# B&R Automation Studio project mappFramework
Automation Studio 4.12.4.107 SP; technology packages: mapp 5.18.0, mappCockpit 5.18.0, mappMotion 5.18.1, mappView 5.18.1

## Configuration Simulation

CPU PC_any, AutomationRuntime E4.91, Build 6.3.0, Safety 0.0, Vc V4.72.3

### Task classes (Cpu.sw)
```
Cyclic#1 (cycle 10000 us):
  AlarmMgr <- Infrastructure.VC4.AlarmX.AlarmMgr.prg
  AppAxis_1 <- MachineControl.AppAxis_1.AppAxis_1.prg
  AxisMgr <- MachineControl.AxisTemplate.AxisMgr.prg [disabled]
Cyclic#8 (cycle 10000 us):
  BackupMgr <- Infrastructure.VC4.Backup.BackupMgr.prg
  FileMgr <- Infrastructure.VC4.File.FileMgr.prg
  UsbMgr <- Infrastructure.VC4.Usb.UsbMgr.prg  // USB manager
  RecipeMgr <- Infrastructure.VC4.Recipe.RecipeMgr.prg
  UserXMgr <- Infrastructure.VC4.UserX.UserXMgr.prg
  AuditMgr <- Infrastructure.VC4.Audit.AuditMgr.prg
  ReportMgr <- Infrastructure.VC4.Report.ReportMgr.prg
NcDataObjects: McDriveLog
VcDataObjects: mappFr <- VC4.mappFrameworkVisu.dob
Binaries: arsvcreg, mCoWebSc, McProfGen, mcacpdrv, TCLang, arflatprv, FWRules, arcoal, udbdef, mvLoader, TCData, vcfntttf, vcxml, vccbmp, vcshared, vccscale, vcmgr, vccshape, vcfile, vcgclass, vccpiech, arial, vcchspot, vccslider, vcdsint, vccbtn, vccline, vcpfar00, vccovl, vcctext, vcalarm, vcbclass, vcrt, vccnum, vccstr, Visu03, vccddbox, arialbd, vcctrend, vcpdsw, vccpopup, vccurl, vcnet, vcpdvnc, vcdsloc, vcclbox, Visu02, Visu01, vctcal, vcchtml, vccdt, vcpkat, UserXCfg, UserXlogin, arconfig, FileCfg, RecipeXML, TC, RecipeFile, User, AlarmXCfg, asfw, iomap, Role, Axis1Alm, VAppAxis1, ashwd, RecipeCSV, Settings, AppAxis1, BackupCfg, ashwac, AlarmXHist, sysconf, Axis1Grp, BackupFile, AuditCfg, UnitCfg, CustomCfg, AdvCfg, ReportFile, SimpleCfg, MachineGrp
Libraries: runtime, astime, FileIO, AsBrStr, MpBase, MpAlarmX, MpServer, sys_lib, standard, AsZip, CoTrace, MpAxis, MpRecipe, MpCom, McAxis, McBase, McAcpAx, McPureVAx, McAcpPar, AsIODiag, MpFile, MpBackup, AsUSB, MpUserX, AsARCfg, IecCheck, MpAudit, MpReport, asieccon, brsystem, aseth, ashw, powerlnk, dataobj, arssl, arproject, arcert, aruser, asepl, vcresman
```

### Hardware
```
PC : PC_any v1.1.1.0 (OrderNumber=PC)
  ConfigurationID = mappFramework516_Simulation
  UserPartitionSize = 256
  Cyclic1Duration = 10000
  Cyclic1Stack = 32000
  Cyclic5Duration = 10000
  Cyclic8Duration = 10000
  Cyclic8Stack = 32000
  FileDevice1
  FileDeviceName1 = USER
  FileDevicePath1 = USER_PATH
  FileDevice2
  FileDeviceName2 = mappAlarmXFiles
  FileDevicePath2 = USER_PATH:\AlarmX
  FileDevice3
  FileDeviceName3 = mappBackupFiles
  FileDevicePath3 = USER_PATH:\Backup
  FileDevice4
  FileDeviceName4 = mappRecipeFiles
  FileDevicePath4 = USER_PATH:\Recipe
  FileDevice5
  FileDeviceName5 = mappUserXFiles
  FileDevicePath5 = USER_PATH:\UserX
  FileDevice6
  FileDeviceName6 = mappAuditFiles
  FileDevicePath6 = USER_PATH:\Audit
  FileDevice7
  FileDeviceName7 = mappDataFiles
  FileDevicePath7 = USER_PATH:\Data
  FileDevice8
  FileDeviceName8 = mappReportFiles
  FileDevicePath8 = USER_PATH:\Report
  FileDevice9
  FileDeviceName9 = mappPackMLFiles
  FileDevicePath9 = USER_PATH:\PackML
  FtpUser1
  FtpUsername1 = Admin
  FtpUserPassword1 = jhTZ9rja+dMo4uQziZxIvYZJ7RF3iWJ9y9zyiFMZfoo=  // 123ABc
  FtpUserSalt1 = 8r0jnJ0m
  FTPAccessRight1 = 0
  FTPdevice1 = ALL
  ActivateOpcUa = 1
  OpcUaActivateAuditEvents = 1
  OpcUa_Security_AdminRole = Administrators
  OpcUaInformationModels_PV_Version = 1
```

### VAppAxis1.purevaxcfg - PC/mappMotion/AppAxis_1/VAppAxis1.purevaxcfg
```
Element gMpLinkPureVAxCfgAppAxis_1 (Type=purevaxcfg)
  TypeID = PureVAxConfig
  PureVAxis:
    AxisReference = gMpLinkAppAxis_1
    Homing:
      Mode = RestorePosition
      RestorePositionVariable = ::AxisMgr:RestorePosition
    JerkFilter = NotUsed
```

### AlarmXCfg.mpalarmxcore - PC/mappServices/AlarmX/AlarmXCfg.mpalarmxcore
```
Element gMpLinkAlarmXCore (Type=mpalarmxcore)
  mapp.AlarmX.Core:
    BySeverity:
      [0]:
        Severity = 1..9
        [0] = Reaction
          Name = Info
      [1]:
        Severity = 10..19
        [0] = Reaction
          Name = Warning
      [2]:
        Severity = 20..29
        [0] = Reaction
          Name = Error
  mapp.AlarmX.Core.Configuration:
    [0]:
      Name = EmergencyStop_0
      Message = {$mappFramework/AlarmX/Alarms/EmergencyStop.0}
      Severity = 29
      Behavior = DiscreteValueMonitoring
        Monitoring:
          MonitoredPV = ::AlarmMgr:SafetyInputs.EmergencyStop[0]
          TriggerValues:
            [0] = 1
    [1]:
      Name = EmergencyStop_1
      Message = {$mappFramework/AlarmX/Alarms/EmergencyStop.1}
      Behavior = DiscreteValueMonitoring
        Monitoring:
          MonitoredPV = ::AlarmMgr:SafetyInputs.EmergencyStop[1]
          TriggerValues:
            [0] = 1
    [2]:
      Name = EmergencyStop_2
      Message = {$mappFramework/AlarmX/Alarms/EmergencyStop.2}
      Behavior = DiscreteValueMonitoring
        Monitoring:
          MonitoredPV = ::AlarmMgr:SafetyInputs.EmergencyStop[2]
          TriggerValues:
            [0] = 1
    [3]:
      Name = SafetyDoor_0
      Message = {$mappFramework/AlarmX/Alarms/SafetyDoor.0}
      Severity = 29
      Behavior = DiscreteValueMonitoring
        Monitoring:
          MonitoredPV = ::AlarmMgr:SafetyInputs.SafetyDoor[0]
          TriggerValues:
            [0] = 1
    [4]:
      Name = SafetyDoor_1
      Message = {$mappFramework/AlarmX/Alarms/SafetyDoor.1}
      Severity = 29
      Behavior = DiscreteValueMonitoring
        Monitoring:
          MonitoredPV = ::AlarmMgr:SafetyInputs.SafetyDoor[1]
          TriggerValues:
            [0] = 1
    [5]:
      Name = SafetyDoor_2
      Message = {$mappFramework/AlarmX/Alarms/SafetyDoor.2}
      Severity = 29
      Behavior = DiscreteValueMonitoring
        Monitoring:
          MonitoredPV = ::AlarmMgr:SafetyInputs.SafetyDoor[2]
          TriggerValues:
            [0] = 1
    [6]:
      Name = SafetyDoor_3
      Message = {$mappFramework/AlarmX/Alarms/SafetyDoor.3}
      Severity = 29
      Behavior = DiscreteValueMonitoring
        Monitoring:
          MonitoredPV = ::AlarmMgr:SafetyInputs.SafetyDoor[3]
          TriggerValues:
            [0] = 1
    [7]:
      Name = SafetyDoor_4
      Message = {$mappFramework/AlarmX/Alarms/SafetyDoor.4}
      Severity = 29
      Behavior = DiscreteValueMonitoring
        Monitoring:
          MonitoredPV = ::AlarmMgr:SafetyInputs.SafetyDoor[4]
          TriggerValues:
            [0] = 1
    [8]:
      Name = SafetyDoor_5
      Message = {$mappFramework/AlarmX/Alarms/SafetyDoor.5}
      Severity = 29
      Behavior = DiscreteValueMonitoring
        Monitoring:
          MonitoredPV = ::AlarmMgr:SafetyInputs.SafetyDoor[5]
          TriggerValues:
            [0] = 1
    [9]:
      Name = LevelMonitoringExample
      Message = {$mappFramework/AlarmX/Alarms/LevelMonitoringAlarmExample} {=$mappFramework/AlarmX/Alarms/{&LimitText}}
      Behavior = LevelMonitoring
        Monitoring:
          MonitoredPV = ::AlarmMgr:AlarmExamples.LevelMonitoring
          LowLimitEnable = Static
            Limit = 20
            LimitText = LevelMonitoringAlarmLowTextExample
            LowLowLimitEnable = Static
              Limit = 10
              LimitText = LevelMonitoringAlarmLowLowTextExample
          HighLimitEnable = Static
            Limit = 80
            LimitText = LevelMonitoringAlarmHighTextExample
            HighHighLimitEnable = Static
              Limit = 90
              LimitText = LevelMonitoringAlarmHighHighTextExample
    [10]:
      Name = DeviationMonitoringExample
      Message = {$mappFramework/AlarmX/Alarms/DeviationMonitoringAlarmExample} {&LimitText}
      Behavior = DeviationMonitoring
        Monitoring:
          MonitoredPV = ::AlarmMgr:AlarmExamples.DeviationMonitoring
          SetpointPV = ::AlarmMgr:AlarmExamples.DeviationMonitoringSetpoint
          LowLimitEnable = Static
            Limit = -5
            LimitText = Low limit exceeded
          HighLimitEnable = Static
            Limit = 5
            LimitText = High limit exceeded
    [11]:
      Name = RateOfChangeExample
      Message = {$mappFramework/AlarmX/Alarms/RateOfChangeAlarmExample}
      Behavior = RateOfChangeMonitoring
        Monitoring:
          MonitoredPV = ::AlarmMgr:AlarmExamples.RateOfChange
          HighLimitEnable = Static
            Limit = 5
            LimitText = High limit exceeded
    [12]:
      Name = SnippetExample
      Message = Show a snippet directly: {&snippet1}. Show from localizable text: {$mappFramework/AlarmX/Alarms/SnippetExample}
      Behavior = DiscreteValueMonitoring
        Monitoring:
          MonitoredPV = ::AlarmMgr:AlarmExamples.SnippetValue
          TriggerValues:
            [0] = 50..100
    [13]:
      Name = MpAlarmXControlExample
      Message = {$mappFramework/AlarmX/Alarms/MpAlarmXControlExample}
      Severity = 20
      Behavior:
        Async = TRUE
    [14]:
      Name = Alarm0
      Message = {$mappFramework/AlarmX/Alarms/Alarm.0}
      Behavior = DiscreteValueMonitoring
        Monitoring:
          MonitoredPV = ::AlarmMgr:Alarms[0]
          InhibitPV = ::AlarmMgr:CommissioningModeActive
          TriggerValues:
            [0] = 1
    [15]:
      Name = Alarm1
      Message = {$mappFramework/AlarmX/Alarms/Alarm.1}
      Code = 1
      Behavior = DiscreteValueMonitoring
        Monitoring:
          MonitoredPV = ::AlarmMgr:Alarms[1]
          TriggerValues:
            [0] = 1
    [16]:
      Name = Alarm2
      Message = {$mappFramework/AlarmX/Alarms/Alarm.2}
      Code = 2
      Behavior = DiscreteValueMonitoring
        Monitoring:
          MonitoredPV = ::AlarmMgr:Alarms[2]
          TriggerValues:
            [0] = 1
    [17]:
      Name = Alarm3
      Message = {$mappFramework/AlarmX/Alarms/Alarm.3}
      Code = 3
      Behavior = DiscreteValueMonitoring
        Monitoring:
          MonitoredPV = ::AlarmMgr:Alarms[3]
          TriggerValues:
            [0] = 1
    [18]:
      Name = Alarm4
      Message = {$mappFramework/AlarmX/Alarms/Alarm.4}
      Code = 4
      Behavior = DiscreteValueMonitoring
        Monitoring:
          MonitoredPV = ::AlarmMgr:Alarms[4]
          TriggerValues:
            [0] = 1
    [19]:
      Name = Alarm5
      Message = {$mappFramework/AlarmX/Alarms/Alarm.5}
      Code = 5
      Behavior = DiscreteValueMonitoring
        Monitoring:
          MonitoredPV = ::AlarmMgr:Alarms[5]
          TriggerValues:
            [0] = 1
    [20]:
      Name = Alarm6
      Message = {$mappFramework/AlarmX/Alarms/Alarm.6}
      Code = 6
      Behavior = DiscreteValueMonitoring
        Monitoring:
          MonitoredPV = ::AlarmMgr:Alarms[6]
          TriggerValues:
            [0] = 1
    [21]:
      Name = Alarm7
      Message = {$mappFramework/AlarmX/Alarms/Alarm.7}
      Code = 7
      Behavior = DiscreteValueMonitoring
        Monitoring:
          MonitoredPV = ::AlarmMgr:Alarms[7]
          TriggerValues:
            [0] = 1
    [22]:
      Name = Alarm8
      Message = {$mappFramework/AlarmX/Alarms/Alarm.8}
      Code = 8
      Behavior = DiscreteValueMonitoring
        Monitoring:
          MonitoredPV = ::AlarmMgr:Alarms[8]
          TriggerValues:
            [0] = 1
    [23]:
      Name = Alarm9
      Message = {$mappFramework/AlarmX/Alarms/Alarm.9}
      Code = 9
      Behavior = DiscreteValueMonitoring
        Monitoring:
          MonitoredPV = ::AlarmMgr:Alarms[9]
          TriggerValues:
            [0] = 1
    [24]:
      Name = Alarm10
      Message = {$mappFramework/AlarmX/Alarms/Alarm.10}
      Code = 10
      Behavior = DiscreteValueMonitoring
        Monitoring:
          MonitoredPV = ::AlarmMgr:Alarms[10]
          TriggerValues:
            [0] = 1
    [25]:
      Name = Alarm11
      Message = {$mappFramework/AlarmX/Alarms/Alarm.11}
      Code = 11
      Behavior = DiscreteValueMonitoring
        Monitoring:
          MonitoredPV = ::AlarmMgr:Alarms[11]
          TriggerValues:
            [0] = 1
    [26]:
      Name = Alarm12
      Message = {$mappFramework/AlarmX/Alarms/Alarm.12}
      Code = 12
      Behavior = DiscreteValueMonitoring
        Monitoring:
          MonitoredPV = ::AlarmMgr:Alarms[12]
          TriggerValues:
            [0] = 1
    [27]:
      Name = Alarm13
      Message = {$mappFramework/AlarmX/Alarms/Alarm.13}
      Code = 13
      Behavior = DiscreteValueMonitoring
        Monitoring:
          MonitoredPV = ::AlarmMgr:Alarms[13]
          TriggerValues:
            [0] = 1
    [28]:
      Name = Alarm14
      Message = {$mappFramework/AlarmX/Alarms/Alarm.14}
      Code = 14
      Behavior = DiscreteValueMonitoring
        Monitoring:
          MonitoredPV = ::AlarmMgr:Alarms[14]
          TriggerValues:
            [0] = 1
    [29]:
      Name = Alarm15
      Message = {$mappFramework/AlarmX/Alarms/Alarm.15}
      Code = 15
      Behavior = DiscreteValueMonitoring
        Monitoring:
          MonitoredPV = ::AlarmMgr:Alarms[15]
          TriggerValues:
            [0] = 1
    [30]:
      Name = Alarm16
      Message = {$mappFramework/AlarmX/Alarms/Alarm.16}
      Code = 16
      Behavior = DiscreteValueMonitoring
        Monitoring:
          MonitoredPV = ::AlarmMgr:Alarms[16]
          TriggerValues:
            [0] = 1
    [31]:
      Name = Alarm17
      Message = {$mappFramework/AlarmX/Alarms/Alarm.17}
      Code = 17
      Behavior = DiscreteValueMonitoring
        Monitoring:
          MonitoredPV = ::AlarmMgr:Alarms[17]
          TriggerValues:
            [0] = 1
    [32]:
      Name = Alarm18
      Message = {$mappFramework/AlarmX/Alarms/Alarm.18}
      Code = 18
      Behavior = DiscreteValueMonitoring
        Monitoring:
          MonitoredPV = ::AlarmMgr:Alarms[18]
          TriggerValues:
            [0] = 1
    [33]:
      Name = Alarm19
      Message = {$mappFramework/AlarmX/Alarms/Alarm.19}
      Code = 19
      Behavior = DiscreteValueMonitoring
        Monitoring:
          MonitoredPV = ::AlarmMgr:Alarms[19]
          TriggerValues:
            [0] = 1
    [34]:
      Name = Alarm20
      Message = {$mappFramework/AlarmX/Alarms/Alarm.20}
      Behavior = DiscreteValueMonitoring
        Monitoring:
          MonitoredPV = ::AlarmMgr:Alarms[20]
          TriggerValues:
            [0] = 1
    [35]:
      Name = Alarm21
      Message = {$mappFramework/AlarmX/Alarms/Alarm.21}
      Code = 21
      Behavior = DiscreteValueMonitoring
        Monitoring:
          MonitoredPV = ::AlarmMgr:Alarms[21]
          TriggerValues:
            [0] = 1
    [36]:
      Name = Alarm22
      Message = {$mappFramework/AlarmX/Alarms/Alarm.22}
      Code = 22
      Behavior = DiscreteValueMonitoring
        Monitoring:
          MonitoredPV = ::AlarmMgr:Alarms[22]
          TriggerValues:
            [0] = 1
    [37]:
      Name = Alarm23
      Message = {$mappFramework/AlarmX/Alarms/Alarm.23}
      Code = 23
      Behavior = DiscreteValueMonitoring
        Monitoring:
          MonitoredPV = ::AlarmMgr:Alarms[23]
          TriggerValues:
            [0] = 1
    [38]:
      Name = Alarm24
      Message = {$mappFramework/AlarmX/Alarms/Alarm.24}
      Code = 24
      Behavior = DiscreteValueMonitoring
        Monitoring:
          MonitoredPV = ::AlarmMgr:Alarms[24]
          TriggerValues:
            [0] = 1
    [39]:
      Name = Alarm25
      Message = {$mappFramework/AlarmX/Alarms/Alarm.25}
      Code = 25
      Behavior = DiscreteValueMonitoring
        Monitoring:
          MonitoredPV = ::AlarmMgr:Alarms[25]
          TriggerValues:
            [0] = 1
    [40]:
      Name = Alarm26
      Message = {$mappFramework/AlarmX/Alarms/Alarm.26}
      Code = 26
      Behavior = DiscreteValueMonitoring
        Monitoring:
          MonitoredPV = ::AlarmMgr:Alarms[26]
          TriggerValues:
            [0] = 1
    [41]:
      Name = Alarm27
      Message = {$mappFramework/AlarmX/Alarms/Alarm.27}
      Code = 27
      Behavior = DiscreteValueMonitoring
        Monitoring:
          MonitoredPV = ::AlarmMgr:Alarms[27]
          TriggerValues:
            [0] = 1
    [42]:
      Name = Alarm28
      Message = {$mappFramework/AlarmX/Alarms/Alarm.28}
      Code = 28
      Behavior = DiscreteValueMonitoring
        Monitoring:
          MonitoredPV = ::AlarmMgr:Alarms[28]
          TriggerValues:
            [0] = 1
    [43]:
      Name = Alarm29
      Message = {$mappFramework/AlarmX/Alarms/Alarm.29}
      Code = 29
      Behavior = DiscreteValueMonitoring
        Monitoring:
          MonitoredPV = ::AlarmMgr:Alarms[29]
          TriggerValues:
            [0] = 1
    [44]:
      Name = Alarm30
      Message = {$mappFramework/AlarmX/Alarms/Alarm.30}
      Behavior = DiscreteValueMonitoring
        Monitoring:
          MonitoredPV = ::AlarmMgr:Alarms[30]
          TriggerValues:
            [0] = 1
    [45]:
      Name = Alarm31
      Message = {$mappFramework/AlarmX/Alarms/Alarm.31}
      Code = 31
      Behavior = DiscreteValueMonitoring
        Monitoring:
          MonitoredPV = ::AlarmMgr:Alarms[31]
          TriggerValues:
            [0] = 1
    [46]:
      Name = Alarm32
      Message = {$mappFramework/AlarmX/Alarms/Alarm.32}
      Code = 32
      Behavior = DiscreteValueMonitoring
        Monitoring:
          MonitoredPV = ::AlarmMgr:Alarms[32]
          TriggerValues:
            [0] = 1
    [47]:
      Name = Alarm33
      Message = {$mappFramework/AlarmX/Alarms/Alarm.33}
      Code = 33
      Behavior = DiscreteValueMonitoring
        Monitoring:
          MonitoredPV = ::AlarmMgr:Alarms[33]
          TriggerValues:
            [0] = 1
    [48]:
      Name = Alarm34
      Message = {$mappFramework/AlarmX/Alarms/Alarm.34}
      Code = 34
      Behavior = DiscreteValueMonitoring
        Monitoring:
          MonitoredPV = ::AlarmMgr:Alarms[34]
          TriggerValues:
            [0] = 1
    [49]:
      Name = Alarm35
      Message = {$mappFramework/AlarmX/Alarms/Alarm.35}
      Code = 35
      Behavior = DiscreteValueMonitoring
        Monitoring:
          MonitoredPV = ::AlarmMgr:Alarms[35]
          TriggerValues:
            [0] = 1
    [50]:
      Name = Alarm36
      Message = {$mappFramework/AlarmX/Alarms/Alarm.36}
      Code = 36
      Behavior = DiscreteValueMonitoring
        Monitoring:
          MonitoredPV = ::AlarmMgr:Alarms[36]
          TriggerValues:
            [0] = 1
    [51]:
      Name = Alarm37
      Message = {$mappFramework/AlarmX/Alarms/Alarm.37}
      Code = 37
      Behavior = DiscreteValueMonitoring
        Monitoring:
          MonitoredPV = ::AlarmMgr:Alarms[37]
          TriggerValues:
            [0] = 1
    [52]:
      Name = Alarm38
      Message = {$mappFramework/AlarmX/Alarms/Alarm.38}
      Code = 38
      Behavior = DiscreteValueMonitoring
        Monitoring:
          MonitoredPV = ::AlarmMgr:Alarms[38]
          TriggerValues:
            [0] = 1
    [53]:
      Name = Alarm39
      Message = {$mappFramework/AlarmX/Alarms/Alarm.39}
      Code = 39
      Behavior = DiscreteValueMonitoring
        Monitoring:
          MonitoredPV = ::AlarmMgr:Alarms[39]
          TriggerValues:
            [0] = 1
    [54]:
      Name = Alarm40
      Message = {$mappFramework/AlarmX/Alarms/Alarm.40}
      Behavior = DiscreteValueMonitoring
        Monitoring:
          MonitoredPV = ::AlarmMgr:Alarms[40]
          TriggerValues:
            [0] = 1
    [55]:
      Name = Alarm41
      Message = {$mappFramework/AlarmX/Alarms/Alarm.41}
      Code = 41
      Behavior = DiscreteValueMonitoring
        Monitoring:
          MonitoredPV = ::AlarmMgr:Alarms[41]
          TriggerValues:
            [0] = 1
    [56]:
      Name = Alarm42
      Message = {$mappFramework/AlarmX/Alarms/Alarm.42}
      Code = 42
      Behavior = DiscreteValueMonitoring
        Monitoring:
          MonitoredPV = ::AlarmMgr:Alarms[42]
          TriggerValues:
            [0] = 1
    [57]:
      Name = Alarm43
      Message = {$mappFramework/AlarmX/Alarms/Alarm.43}
      Code = 43
      Behavior = DiscreteValueMonitoring
        Monitoring:
          MonitoredPV = ::AlarmMgr:Alarms[43]
          TriggerValues:
            [0] = 1
    [58]:
      Name = Alarm44
      Message = {$mappFramework/AlarmX/Alarms/Alarm.44}
      Code = 44
      Behavior = DiscreteValueMonitoring
        Monitoring:
          MonitoredPV = ::AlarmMgr:Alarms[44]
          TriggerValues:
            [0] = 1
    [59]:
      Name = Alarm45
      Message = {$mappFramework/AlarmX/Alarms/Alarm.45}
      Code = 45
      Behavior = DiscreteValueMonitoring
        Monitoring:
          MonitoredPV = ::AlarmMgr:Alarms[45]
          TriggerValues:
            [0] = 1
    [60]:
      Name = Alarm46
      Message = {$mappFramework/AlarmX/Alarms/Alarm.46}
      Code = 46
      Behavior = DiscreteValueMonitoring
        Monitoring:
          MonitoredPV = ::AlarmMgr:Alarms[46]
          TriggerValues:
            [0] = 1
    [61]:
      Name = Alarm47
      Message = {$mappFramework/AlarmX/Alarms/Alarm.47}
      Code = 47
      Behavior = DiscreteValueMonitoring
        Monitoring:
          MonitoredPV = ::AlarmMgr:Alarms[47]
          TriggerValues:
            [0] = 1
    [62]:
      Name = Alarm48
      Message = {$mappFramework/AlarmX/Alarms/Alarm.48}
      Code = 48
      Behavior = DiscreteValueMonitoring
        Monitoring:
          MonitoredPV = ::AlarmMgr:Alarms[48]
          TriggerValues:
            [0] = 1
    [63]:
      Name = Alarm49
      Message = {$mappFramework/AlarmX/Alarms/Alarm.49}
      Code = 49
      Behavior = DiscreteValueMonitoring
        Monitoring:
          MonitoredPV = ::AlarmMgr:Alarms[49]
          TriggerValues:
            [0] = 1
    [64]:
      Name = Alarm50
      Message = {$mappFramework/AlarmX/Alarms/Alarm.50}
      Behavior = DiscreteValueMonitoring
        Monitoring:
          MonitoredPV = ::AlarmMgr:Alarms[50]
          TriggerValues:
            [0] = 1
    [65]:
      Name = Alarm51
      Message = {$mappFramework/AlarmX/Alarms/Alarm.51}
      Code = 51
      Behavior = DiscreteValueMonitoring
        Monitoring:
          MonitoredPV = ::AlarmMgr:Alarms[51]
          TriggerValues:
            [0] = 1
    [66]:
      Name = Alarm52
      Message = {$mappFramework/AlarmX/Alarms/Alarm.52}
      Code = 52
      Behavior = DiscreteValueMonitoring
        Monitoring:
          MonitoredPV = ::AlarmMgr:Alarms[52]
          TriggerValues:
            [0] = 1
    [67]:
      Name = Alarm53
      Message = {$mappFramework/AlarmX/Alarms/Alarm.53}
      Code = 53
      Behavior = DiscreteValueMonitoring
        Monitoring:
          MonitoredPV = ::AlarmMgr:Alarms[53]
          TriggerValues:
            [0] = 1
    [68]:
      Name = Alarm54
      Message = {$mappFramework/AlarmX/Alarms/Alarm.54}
      Code = 54
      Behavior = DiscreteValueMonitoring
        Monitoring:
          MonitoredPV = ::AlarmMgr:Alarms[54]
          TriggerValues:
            [0] = 1
    [69]:
      Name = Alarm55
      Message = {$mappFramework/AlarmX/Alarms/Alarm.55}
      Code = 55
      Behavior = DiscreteValueMonitoring
        Monitoring:
          MonitoredPV = ::AlarmMgr:Alarms[55]
          TriggerValues:
            [0] = 1
    [70]:
      Name = Alarm56
      Message = {$mappFramework/AlarmX/Alarms/Alarm.56}
      Code = 56
      Behavior = DiscreteValueMonitoring
        Monitoring:
          MonitoredPV = ::AlarmMgr:Alarms[56]
          TriggerValues:
            [0] = 1
    [71]:
      Name = Alarm57
      Message = {$mappFramework/AlarmX/Alarms/Alarm.57}
      Code = 57
      Behavior = DiscreteValueMonitoring
        Monitoring:
          MonitoredPV = ::AlarmMgr:Alarms[57]
          TriggerValues:
            [0] = 1
    [72]:
      Name = Alarm58
      Message = {$mappFramework/AlarmX/Alarms/Alarm.58}
      Code = 58
      Behavior = DiscreteValueMonitoring
        Monitoring:
          MonitoredPV = ::AlarmMgr:Alarms[58]
          TriggerValues:
            [0] = 1
    [73]:
      Name = Alarm59
      Message = {$mappFramework/AlarmX/Alarms/Alarm.59}
      Code = 59
      Behavior = DiscreteValueMonitoring
        Monitoring:
          MonitoredPV = ::AlarmMgr:Alarms[59]
          TriggerValues:
            [0] = 1
    [74]:
      Name = Alarm60
      Message = {$mappFramework/AlarmX/Alarms/Alarm.60}
      Behavior = DiscreteValueMonitoring
        Monitoring:
          MonitoredPV = ::AlarmMgr:Alarms[60]
          TriggerValues:
            [0] = 1
    [75]:
      Name = Alarm61
      Message = {$mappFramework/AlarmX/Alarms/Alarm.61}
      Code = 61
      Behavior = DiscreteValueMonitoring
        Monitoring:
          MonitoredPV = ::AlarmMgr:Alarms[61]
          TriggerValues:
            [0] = 1
    [76]:
      Name = Alarm62
      Message = {$mappFramework/AlarmX/Alarms/Alarm.62}
      Code = 62
      Behavior = DiscreteValueMonitoring
        Monitoring:
          MonitoredPV = ::AlarmMgr:Alarms[62]
          TriggerValues:
            [0] = 1
    [77]:
      Name = Alarm63
      Message = {$mappFramework/AlarmX/Alarms/Alarm.63}
      Code = 63
      Behavior = DiscreteValueMonitoring
        Monitoring:
          MonitoredPV = ::AlarmMgr:Alarms[63]
          TriggerValues:
            [0] = 1
    [78]:
      Name = Alarm64
      Message = {$mappFramework/AlarmX/Alarms/Alarm.64}
      Code = 64
      Behavior = DiscreteValueMonitoring
        Monitoring:
          MonitoredPV = ::AlarmMgr:Alarms[64]
          TriggerValues:
            [0] = 1
    [79]:
      Name = Alarm65
      Message = {$mappFramework/AlarmX/Alarms/Alarm.65}
      Code = 65
      Behavior = DiscreteValueMonitoring
        Monitoring:
          MonitoredPV = ::AlarmMgr:Alarms[65]
          TriggerValues:
            [0] = 1
    [80]:
      Name = Alarm66
      Message = {$mappFramework/AlarmX/Alarms/Alarm.66}
      Code = 66
      Behavior = DiscreteValueMonitoring
        Monitoring:
          MonitoredPV = ::AlarmMgr:Alarms[66]
          TriggerValues:
            [0] = 1
    [81]:
      Name = Alarm67
      Message = {$mappFramework/AlarmX/Alarms/Alarm.67}
      Code = 67
      Behavior = DiscreteValueMonitoring
        Monitoring:
          MonitoredPV = ::AlarmMgr:Alarms[67]
          TriggerValues:
            [0] = 1
    [82]:
      Name = Alarm68
      Message = {$mappFramework/AlarmX/Alarms/Alarm.68}
      Code = 68
      Behavior = DiscreteValueMonitoring
        Monitoring:
          MonitoredPV = ::AlarmMgr:Alarms[68]
          TriggerValues:
            [0] = 1
    [83]:
      Name = Alarm69
      Message = {$mappFramework/AlarmX/Alarms/Alarm.69}
      Code = 69
      Behavior = DiscreteValueMonitoring
        Monitoring:
          MonitoredPV = ::AlarmMgr:Alarms[69]
          TriggerValues:
            [0] = 1
    [84]:
      Name = Alarm70
      Message = {$mappFramework/AlarmX/Alarms/Alarm.70}
      Behavior = DiscreteValueMonitoring
        Monitoring:
          MonitoredPV = ::AlarmMgr:Alarms[70]
          TriggerValues:
            [0] = 1
    [85]:
      Name = Alarm71
      Message = {$mappFramework/AlarmX/Alarms/Alarm.71}
      Code = 71
      Behavior = DiscreteValueMonitoring
        Monitoring:
          MonitoredPV = ::AlarmMgr:Alarms[71]
          TriggerValues:
            [0] = 1
    [86]:
      Name = Alarm72
      Message = {$mappFramework/AlarmX/Alarms/Alarm.72}
      Code = 72
      Behavior = DiscreteValueMonitoring
        Monitoring:
          MonitoredPV = ::AlarmMgr:Alarms[72]
          TriggerValues:
            [0] = 1
    [87]:
      Name = Alarm73
      Message = {$mappFramework/AlarmX/Alarms/Alarm.73}
      Code = 73
      Behavior = DiscreteValueMonitoring
        Monitoring:
          MonitoredPV = ::AlarmMgr:Alarms[73]
          TriggerValues:
            [0] = 1
    [88]:
      Name = Alarm74
      Message = {$mappFramework/AlarmX/Alarms/Alarm.74}
      Code = 74
      Behavior = DiscreteValueMonitoring
        Monitoring:
          MonitoredPV = ::AlarmMgr:Alarms[74]
          TriggerValues:
            [0] = 1
    [89]:
      Name = Alarm75
      Message = {$mappFramework/AlarmX/Alarms/Alarm.75}
      Code = 75
      Behavior = DiscreteValueMonitoring
        Monitoring:
          MonitoredPV = ::AlarmMgr:Alarms[75]
          TriggerValues:
            [0] = 1
    [90]:
      Name = Alarm76
      Message = {$mappFramework/AlarmX/Alarms/Alarm.76}
      Code = 76
      Behavior = DiscreteValueMonitoring
        Monitoring:
          MonitoredPV = ::AlarmMgr:Alarms[76]
          TriggerValues:
            [0] = 1
    [91]:
      Name = Alarm77
      Message = {$mappFramework/AlarmX/Alarms/Alarm.77}
      Code = 77
      Behavior = DiscreteValueMonitoring
        Monitoring:
          MonitoredPV = ::AlarmMgr:Alarms[77]
          TriggerValues:
            [0] = 1
    [92]:
      Name = Alarm78
      Message = {$mappFramework/AlarmX/Alarms/Alarm.78}
      Code = 78
      Behavior = DiscreteValueMonitoring
        Monitoring:
          MonitoredPV = ::AlarmMgr:Alarms[78]
          TriggerValues:
            [0] = 1
    [93]:
      Name = Alarm79
      Message = {$mappFramework/AlarmX/Alarms/Alarm.79}
      Code = 79
      Behavior = DiscreteValueMonitoring
        Monitoring:
          MonitoredPV = ::AlarmMgr:Alarms[79]
          TriggerValues:
            [0] = 1
    [94]:
      Name = Alarm80
      Message = {$mappFramework/AlarmX/Alarms/Alarm.80}
      Behavior = DiscreteValueMonitoring
        Monitoring:
          MonitoredPV = ::AlarmMgr:Alarms[80]
          TriggerValues:
            [0] = 1
    [95]:
      Name = Alarm81
      Message = {$mappFramework/AlarmX/Alarms/Alarm.81}
      Code = 81
      Behavior = DiscreteValueMonitoring
        Monitoring:
          MonitoredPV = ::AlarmMgr:Alarms[81]
          TriggerValues:
            [0] = 1
    [96]:
      Name = Alarm82
      Message = {$mappFramework/AlarmX/Alarms/Alarm.82}
      Code = 82
      Behavior = DiscreteValueMonitoring
        Monitoring:
          MonitoredPV = ::AlarmMgr:Alarms[82]
          TriggerValues:
            [0] = 1
    [97]:
      Name = Alarm83
      Message = {$mappFramework/AlarmX/Alarms/Alarm.83}
      Code = 83
      Behavior = DiscreteValueMonitoring
        Monitoring:
          MonitoredPV = ::AlarmMgr:Alarms[83]
          TriggerValues:
            [0] = 1
    [98]:
      Name = Alarm84
      Message = {$mappFramework/AlarmX/Alarms/Alarm.84}
      Code = 84
      Behavior = DiscreteValueMonitoring
        Monitoring:
          MonitoredPV = ::AlarmMgr:Alarms[84]
          TriggerValues:
            [0] = 1
    [99]:
      Name = Alarm85
      Message = {$mappFramework/AlarmX/Alarms/Alarm.85}
      Code = 85
      Behavior = DiscreteValueMonitoring
        Monitoring:
          MonitoredPV = ::AlarmMgr:Alarms[85]
          TriggerValues:
            [0] = 1
    [100]:
      Name = Alarm86
      Message = {$mappFramework/AlarmX/Alarms/Alarm.86}
      Code = 86
      Behavior = DiscreteValueMonitoring
        Monitoring:
          MonitoredPV = ::AlarmMgr:Alarms[86]
          TriggerValues:
            [0] = 1
    [101]:
      Name = Alarm87
      Message = {$mappFramework/AlarmX/Alarms/Alarm.87}
      Code = 87
      Behavior = DiscreteValueMonitoring
        Monitoring:
          MonitoredPV = ::AlarmMgr:Alarms[87]
          TriggerValues:
            [0] = 1
    [102]:
      Name = Alarm88
      Message = {$mappFramework/AlarmX/Alarms/Alarm.88}
      Code = 88
      Behavior = DiscreteValueMonitoring
        Monitoring:
          MonitoredPV = ::AlarmMgr:Alarms[88]
          TriggerValues:
            [0] = 1
    [103]:
      Name = Alarm89
      Message = {$mappFramework/AlarmX/Alarms/Alarm.89}
      Code = 89
      Behavior = DiscreteValueMonitoring
        Monitoring:
          MonitoredPV = ::AlarmMgr:Alarms[89]
          TriggerValues:
            [0] = 1
    [104]:
      Name = Alarm90
      Message = {$mappFramework/AlarmX/Alarms/Alarm.90}
      Behavior = DiscreteValueMonitoring
        Monitoring:
          MonitoredPV = ::AlarmMgr:Alarms[90]
          TriggerValues:
            [0] = 1
    [105]:
      Name = Alarm91
      Message = {$mappFramework/AlarmX/Alarms/Alarm.91}
      Code = 91
      Behavior = DiscreteValueMonitoring
        Monitoring:
          MonitoredPV = ::AlarmMgr:Alarms[91]
          TriggerValues:
            [0] = 1
    [106]:
      Name = Alarm92
      Message = {$mappFramework/AlarmX/Alarms/Alarm.92}
      Code = 92
      Behavior = DiscreteValueMonitoring
        Monitoring:
          MonitoredPV = ::AlarmMgr:Alarms[92]
          TriggerValues:
            [0] = 1
    [107]:
      Name = Alarm93
      Message = {$mappFramework/AlarmX/Alarms/Alarm.93}
      Code = 93
      Behavior = DiscreteValueMonitoring
        Monitoring:
          MonitoredPV = ::AlarmMgr:Alarms[93]
          TriggerValues:
            [0] = 1
    [108]:
      Name = Alarm94
      Message = {$mappFramework/AlarmX/Alarms/Alarm.94}
      Code = 94
      Behavior = DiscreteValueMonitoring
        Monitoring:
          MonitoredPV = ::AlarmMgr:Alarms[94]
          TriggerValues:
            [0] = 1
    [109]:
      Name = Alarm95
      Message = {$mappFramework/AlarmX/Alarms/Alarm.95}
      Code = 95
      Behavior = DiscreteValueMonitoring
        Monitoring:
          MonitoredPV = ::AlarmMgr:Alarms[95]
          TriggerValues:
            [0] = 1
    [110]:
      Name = Alarm96
      Message = {$mappFramework/AlarmX/Alarms/Alarm.96}
      Code = 96
      Behavior = DiscreteValueMonitoring
        Monitoring:
          MonitoredPV = ::AlarmMgr:Alarms[96]
          TriggerValues:
            [0] = 1
    [111]:
      Name = Alarm97
      Message = {$mappFramework/AlarmX/Alarms/Alarm.97}
      Code = 97
      Behavior = DiscreteValueMonitoring
        Monitoring:
          MonitoredPV = ::AlarmMgr:Alarms[97]
          TriggerValues:
            [0] = 1
    [112]:
      Name = Alarm98
      Message = {$mappFramework/AlarmX/Alarms/Alarm.98}
      Code = 98
      Behavior = DiscreteValueMonitoring
        Monitoring:
          MonitoredPV = ::AlarmMgr:Alarms[98]
          TriggerValues:
            [0] = 1
    [113]:
      Name = Alarm99
      Message = {$mappFramework/AlarmX/Alarms/Alarm.99}
      Code = 99
      Behavior = DiscreteValueMonitoring
        Monitoring:
          MonitoredPV = ::AlarmMgr:Alarms[99]
          TriggerValues:
            [0] = 1
  mapp.AlarmX.Core.Snippets:
    AutoDetect = 1
    [0]:
      Key = snippet1
      Value:
        PV = ::AlarmMgr:AlarmExamples.SnippetValue
  mapp.AlarmX.Core.Queries:
    [0]:
      Name = ActiveAlarms
      Update = ::AlarmMgr:AlarmQuery.UpdateCount
      Source:
        SELECT:
          [0]:
            PV = ::AlarmMgr:AlarmQuery.Alarms[].Name
          [1]:
            Column = Message
            PV = ::AlarmMgr:AlarmQuery.Alarms[].Message
          [2]:
            Column = Code
            PV = ::AlarmMgr:AlarmQuery.Alarms[].Code
          [3]:
            Column = Severity
            PV = ::AlarmMgr:AlarmQuery.Alarms[].Severity
          [4]:
            Column = Scope
            PV = ::AlarmMgr:AlarmQuery.Alarms[].Scope
          [5]:
            Column = TimeStamp
            PV = ::AlarmMgr:AlarmQuery.Alarms[].TimeStamp
          [6]:
            Column = AdditionalInformation1
            PV = ::AlarmMgr:AlarmQuery.Alarms[].AdditionalInfo
          [7]:
            Column = StateActive
            PV = ::AlarmMgr:AlarmQuery.Alarms[].Active
          [8]:
            Column = StateAcknowledged
            PV = ::AlarmMgr:AlarmQuery.Alarms[].Acknowledged
```

### AlarmXHist.mpalarmxhistory - PC/mappServices/AlarmX/AlarmXHist.mpalarmxhistory
```
Element gMpLinkAlarmXHistory (Type=mpalarmxhistory)
  mapp.AlarmX.History:
    Memory:
      MemorySize = 6000
    Auditing = MpAudit
    Scope = Branch
```

### Axis1Alm.mpalarmxcore - PC/mappServices/AppAxis_1/Axis1Alm.mpalarmxcore
```
Element gMpLinkAlarmXCoreAppAxis_1 (Type=mpalarmxcore)
  mapp.AlarmX.Core:
    Mapping:
      [0]:
        Alarm = gMpLinkAppAxis_1*
        [0] = Escalate
        [1] = Remain
    BySeverity:
      [0]:
        Severity = 1..9
        [0] = Reaction
          Name = Info
        [1] = Escalate
        [2] = Remain
      [1]:
        Severity = 10..19
        [0] = Reaction
          Name = Warning
        [1] = Escalate
        [2] = Remain
      [2]:
        Severity = 20..29
        [0] = Reaction
          Name = Error
        [1] = Escalate
        [2] = Remain
    Default:
      [0] = Reaction
        Name = Duplicate
      [1] = Escalate
      [2] = Remain
  mapp.AlarmX.Core.Configuration:
    [0]:
      Name = ReferenceRequired
      Message = {$IAT/AppAxis_1/Info/Name} : {$Axis/Alarms/ReferenceRequired}
      Severity = 10
      Behavior = DiscreteValueMonitoring
        Monitoring:
          MonitoredPV = ::AppAxis_1:AxisControl.Status.ReferenceRequired
          TriggerValues:
            [0] = 1
    [1]:
      Name = AppAxis_1SpeedNotSet
      Message = {$IAT/AppAxis_1/Info/Name} : {$Axis/Alarms/AxisSpeedNotSet}
      Code = 250
      Severity = 20
      Behavior:
        Async = TRUE
  mapp.AlarmX.Core.Snippets:
    [0]:
      Key = AxisSpeed
      Value:
        PV = ::AppAxis_1:AxisControl.Parameters.Velocity
```

### AuditCfg.mpaudittrail - PC/mappServices/Audit/AuditCfg.mpaudittrail
```
Element gMpLinkAuditTrail (Type=mpaudittrail)
  Audit:
    Events:
      [0] = 33
      [1] = 2
      [2] = 16
      [3] = 18
      [4] = 113
      [5] = 48
      [6] = 149
    TextSource = TXT
      Name = 
      OutputFormat = MpAudit/Event/Root
    Archive = On
  Alarms = MpAlarmX
```

### CustomCfg.mpaudittrail - PC/mappServices/Audit/CustomCfg.mpaudittrail
```
Element gMpLinkCustomEvents (Type=mpaudittrail)
  Audit:
    Events:
      [0] = 18
    TextSource:
      OutputFormat = {&typ} - {&msg} - {&cmt}
  Alarms = MpAlarmX
```

### UnitCfg.mpcomunit - PC/mappServices/Audit/UnitCfg.mpcomunit
```
Element gGroup (Type=mpcomunit)
  Display:
    Datapoints:
      0:
        Id = ::AuditMgr:HmiAudit.Parameters.SampleVariable
        DisplayUnits:
          Metric:
            Code = CEL
          Imperial:
            Code = FAH
          ImperialUS:
            Code = FAH
    Units:
      0:
        EngineeringUnit:
          Code = CEL
        DisplayUnits:
          Metric:
            Code = CEL
          Imperial:
            Code = FAH
          ImperialUS:
            Code = FAH
```

### BackupCfg.mpbackupcore - PC/mappServices/Backup/BackupCfg.mpbackupcore
```
Element gMpLinkBackupCore (Type=mpbackupcore)
  Backup:
    AutomaticBackup = Enabled
      Mode = Weekly
      OverwriteOldest = Enabled
        MaximumNumberOfBackups = 5
    AutomaticUpdate = Notify
      DeviceName = mappBackupFiles
      Check:
        Time = 57600000
    Auditing = MpAudit
  Alarms = MpAlarmX
```

### BackupFile.mpfilemanagerui - PC/mappServices/Backup/BackupFile.mpfilemanagerui
```
Element gMpLinkFileManagerUIBackup (Type=mpfilemanagerui)
  Alarms = MpAlarmX
    mapp.AlarmX.Core.Configuration:
      [0]:
        Message = {$mappFramework/File/Alarms/DeviceNotFound}
      [1]:
        Message = {$mappFramework/File/Alarms/AlreadyExisting}
      [2]:
        Message = {$mappFramework/File/Alarms/FileSystemError}
```

### Config.mpfilemanager - PC/mappServices/File/Config.mpfilemanager
```
Element FileManagement (Type=mpfilemanager)
  FileManager:
    Auditing = MpAudit
```

### FileCfg.mpfilemanagerui - PC/mappServices/File/FileCfg.mpfilemanagerui
```
Element gMpLinkFileManagerUIFile (Type=mpfilemanagerui)
  Alarms = MpAlarmX
    mapp.AlarmX.Core.Configuration:
      [0]:
        Message = {$mappFramework/File/Alarms/DeviceNotFound}
      [1]:
        Message = {$mappFramework/File/Alarms/AlreadyExisting}
      [2]:
        Message = {$mappFramework/File/Alarms/FileSystemError}
Element gMpLinkFileManagerUIFile_FIFO (Type=mpfilemanagerui)
  Alarms = MpAlarmX
    mapp.AlarmX.Core.Configuration:
      [0]:
        Message = {$mappFramework/File/Alarms/DeviceNotFound}
      [1]:
        Message = {$mappFramework/File/Alarms/AlreadyExisting}
      [2]:
        Message = {$mappFramework/File/Alarms/FileSystemError}
```

### PackMLCfg.mppackmlcore - PC/mappServices/PackML/PackMLCfg.mppackmlcore
```
Element gMpLinkPackMLCore (Type=mppackmlcore)
  Modes:
    Mode[1]:
      ModeID = 1
      Name = Production
```

### PackMLMain.mppackmlmodule - PC/mappServices/PackML/PackMLMain.mppackmlmodule
```
Element gMpPackMLModuleMain (Type=mppackmlmodule)
  Module:
    Name = Main
    Parent = 1
      Unit = gMpLinkPackMLCore
      Activation = 0
```

### RecipeCSV.mprecipecsv - PC/mappServices/Recipe/RecipeCSV.mprecipecsv
```
Element gMpLinkRecipeCsv (Type=mprecipecsv)
  mapp.Recipe.Csv:
    Auditing = MpAudit
  Alarms = MpAlarmX
    mapp.AlarmX.Core.Configuration:
      [0]:
        Message = {$mappFramework/Recipe/Alarms/SaveFailed}
      [1]:
        Message = {$mappFramework/Recipe/Alarms/SaveFailedPartial}
      [2]:
        Message = {$mappFramework/Recipe/Alarms/LoadFailed}
      [3]:
        Message = {$mappFramework/Recipe/Alarms/LoadFailedPartial}
```

### RecipeFile.mpfilemanagerui - PC/mappServices/Recipe/RecipeFile.mpfilemanagerui
```
Element gMpLinkFileManagerUIRecipe (Type=mpfilemanagerui)
  Alarms = MpAlarmX
    mapp.AlarmX.Core.Configuration:
      [0]:
        Message = {$mappFramework/File/Alarms/DeviceNotFound}
      [1]:
        Message = {$mappFramework/File/Alarms/AlreadyExisting}
      [2]:
        Message = {$mappFramework/File/Alarms/FileSystemError}
```

### RecipeXML.mprecipexml - PC/mappServices/Recipe/RecipeXML.mprecipexml
```
Element gMpLinkRecipeXml (Type=mprecipexml)
  mapp.Recipe.Xml:
    Auditing = MpAudit
  Alarms = MpAlarmX
    mapp.AlarmX.Core.Configuration:
      [0]:
        Message = {$mappFramework/Recipe/Alarms/SaveFailed}
      [1]:
        Message = {$mappFramework/Recipe/Alarms/SaveFailedPartial}
        Disable = TRUE
      [2]:
        Message = {$mappFramework/Recipe/Alarms/LoadFailed}
      [3]:
        Message = {$mappFramework/Recipe/Alarms/LoadFailedPartial}
        Disable = TRUE
```

### AdvCfg.mpreportcore - PC/mappServices/Report/AdvCfg.mpreportcore
```
Element gMpLinkAdvancedReport (Type=mpreportcore)
  MpReport:
    Settings:
      ResourceDeviceName = mappReportFiles
      LanguageDependent:
        [0]:
          Language = en
        [1]:
          Language = de
        [2]:
          Language = zh
          Font = 4
    PageLayouts:
      [0]:
        Name = Default
        Orientation = 2
        Margins = 2
    Styles:
      Text:
        [0]:
          Name = Default
        [1]:
          Name = Title
          Size = 20
        [2]:
          Name = Description
          Color = FF9900
        [3]:
          Name = TableText
          NumberOfDecimalPlaces = 2
        [4]:
          Name = ChartText
          NumberOfDecimalPlaces = 2
      Table:
        [0]:
          Name = Default
        [1]:
          Name = ThickBorder_Blue_HighPadding
          BorderWidth = 3
          Color = 0000FF
          Padding = 3
      Line:
        [0]:
          Name = Default
        [1]:
          Name = ThickOrangeLine
          Width = 5
          Color = FF9900
      Chart:
        PieChart:
          [0]:
            Name = Default
          [1]:
            Name = ColorPieChart
            BackColor = 008080
            BorderWidth = 3
            BorderColor = 33CC00
            Padding = 3
        LineChart:
          [0]:
            Name = Default
          [1]:
            Name = ColorLineChart
            BackColor = 008080
            BorderWidth = 3
            BorderColor = 33CC00
            Padding = 3
            GraphBackColor = C0C0C0
            GraphBorderWidth = 3
            GraphBorderColor = 808000
            GridLineWidth = 3
            GridLineColor = 7F7F7F
        BarChart:
          [0]:
            Name = Default
          [1]:
            Name = ColorBarChart
            BackColor = 008080
            BorderWidth = 3
            BorderColor = 33CC00
            Padding = 3
            ItemGapWidth = 3
            GraphBackColor = C0C0C0
            GraphBorderWidth = 3
            GraphBorderColor = 808000
            GridLineWidth = 3
            GridLineColor = 7F7F7F
    Tables:
      [0]:
        Name = DailySummary
        TableStyle = Default
        TextStyle = TableText
        [0]:
          [0] = TextId
            Source = {$mappFramework/Report/Texts/RunTime}
            Width = 20
            HorizontalAlign = 1
          [1] = TextId
            Source = {$mappFramework/Report/Texts/UpTime}
            Width = 20
            HorizontalAlign = 1
          [2] = TextId
            Source = {$mappFramework/Report/Texts/DownTime}
            Width = 20
            HorizontalAlign = 1
          [3] = TextId
            Source = {$mappFramework/Report/Texts/PartsMade}
            Width = 20
            HorizontalAlign = 1
          [4] = TextId
            Source = {$mappFramework/Report/Texts/PPM}
            Width = 10
            HorizontalAlign = 1
          [5] = TextId
            Source = {$mappFramework/Report/Texts/NumRejects}
            Width = 10
            HorizontalAlign = 1
        [1]:
          [0] = ValueId
            Value:
              ProcessVariable = ::ReportMgr:ReportExample.AdvancedReport.OeeLine[0].RunTime
            Width = 20
          [1] = ValueId
            Value:
              ProcessVariable = ::ReportMgr:ReportExample.AdvancedReport.OeeLine[0].UpTime
            Width = 20
          [2] = ValueId
            Value:
              ProcessVariable = ::ReportMgr:ReportExample.AdvancedReport.OeeLine[0].DownTime
            Width = 20
          [3] = ValueId
            Value:
              ProcessVariable = ::ReportMgr:ReportExample.AdvancedReport.OeeLine[0].PartsMade
            Width = 20
            HorizontalAlign = 2
          [4] = ValueId
            Value:
              ProcessVariable = ::ReportMgr:ReportExample.AdvancedReport.OeeLine[0].PPM
            Width = 10
            HorizontalAlign = 2
          [5] = ValueId
            Value:
              ProcessVariable = ::ReportMgr:ReportExample.AdvancedReport.OeeLine[0].NumRejects
            Width = 10
            HorizontalAlign = 2
        [2]:
          [0] = ValueId
            Value:
              ProcessVariable = ::ReportMgr:ReportExample.AdvancedReport.OeeLine[1].RunTime
            Width = 20
          [1] = ValueId
            Value:
              ProcessVariable = ::ReportMgr:ReportExample.AdvancedReport.OeeLine[1].UpTime
            Width = 20
          [2] = ValueId
            Value:
              ProcessVariable = ::ReportMgr:ReportExample.AdvancedReport.OeeLine[1].DownTime
            Width = 20
          [3] = ValueId
            Value:
              ProcessVariable = ::ReportMgr:ReportExample.AdvancedReport.OeeLine[1].PartsMade
            Width = 20
            HorizontalAlign = 2
          [4] = ValueId
            Value:
              ProcessVariable = ::ReportMgr:ReportExample.AdvancedReport.OeeLine[1].PPM
            Width = 10
            HorizontalAlign = 2
          [5] = ValueId
            Value:
              ProcessVariable = ::ReportMgr:ReportExample.AdvancedReport.OeeLine[1].NumRejects
            Width = 10
            HorizontalAlign = 2
        [3]:
          [0] = ValueId
            Value:
              ProcessVariable = ::ReportMgr:ReportExample.AdvancedReport.OeeLine[2].RunTime
            Width = 20
          [1] = ValueId
            Value:
              ProcessVariable = ::ReportMgr:ReportExample.AdvancedReport.OeeLine[2].UpTime
            Width = 20
          [2] = ValueId
            Value:
              ProcessVariable = ::ReportMgr:ReportExample.AdvancedReport.OeeLine[2].DownTime
            Width = 20
          [3] = ValueId
            Value:
              ProcessVariable = ::ReportMgr:ReportExample.AdvancedReport.OeeLine[2].PartsMade
            Width = 20
            HorizontalAlign = 2
          [4] = ValueId
            Value:
              ProcessVariable = ::ReportMgr:ReportExample.AdvancedReport.OeeLine[2].PPM
            Width = 10
            HorizontalAlign = 2
          [5] = ValueId
            Value:
              ProcessVariable = ::ReportMgr:ReportExample.AdvancedReport.OeeLine[2].NumRejects
            Width = 10
            HorizontalAlign = 2
    Charts:
      [0] = LineChart
        Name = TempLineChart
        Heading = SingleText
          Text = {$mappFramework/Report/Texts/TempLineChartHeading}
          HorizontalAlign = 1
          TextStyle = Default
        ChartStyle = Default
        TextStyle = ChartText
        ShowLegend = 4
        Y[0]:
          Name = Temperature
          Label = {$mappFramework/Report/Texts/TempChartYAxisLabel}
          NumberOfGridLines = 9
          GraphMinValue:
            Value = 10
          GraphMaxValue:
            Value = 110
        XAxis:
          ProcessVariable = ::ReportMgr:ReportExample.AdvancedReport.OeeLine[0].TemperatureSample.TimeStamp
        [0]:
          YAxis = Temperature
          Value:
            ProcessVariable = ::ReportMgr:ReportExample.AdvancedReport.OeeLine[0].TemperatureSample.Value
          LegendText = {$mappFramework/Report/Texts/Line1LegendText}
        [1]:
          YAxis = Temperature
          Value:
            ProcessVariable = ::ReportMgr:ReportExample.AdvancedReport.OeeLine[1].TemperatureSample.Value
          LineColor = 33CC00
          LegendText = {$mappFramework/Report/Texts/Line2LegendText}
        [2]:
          YAxis = Temperature
          Value:
            ProcessVariable = ::ReportMgr:ReportExample.AdvancedReport.OeeLine[2].TemperatureSample.Value
          LineColor = 0000FF
          LegendText = {$mappFramework/Report/Texts/Line3LegendText}
      [1] = BarChart
        Name = PartsBarChart
        ChartStyle = Default
        TextStyle = ChartText
        ShowLegend = 4
        YAxis:
          Label = {$mappFramework/Report/Texts/PartsMade}
          NumberOfGridLines = 9
          ItemMaxValue:
            Value = 100000
        [0]:
          Value:
            ProcessVariable = ::ReportMgr:ReportExample.AdvancedReport.OeeLine[0].PartsMade
          ItemColor = 0000FF
          LegendText = {$mappFramework/Report/Texts/Line1LegendText}
        [1]:
          Value:
            ProcessVariable = ::ReportMgr:ReportExample.AdvancedReport.OeeLine[1].PartsMade
          ItemColor = 008080
          LegendText = {$mappFramework/Report/Texts/Line2LegendText}
        [2]:
          Value:
            ProcessVariable = ::ReportMgr:ReportExample.AdvancedReport.OeeLine[2].PartsMade
          ItemColor = 33CC00
          LegendText = {$mappFramework/Report/Texts/Line3LegendText}
      [2] = BarChart
        Name = RejectsBarChart
        ChartStyle = Default
        TextStyle = ChartText
        ShowLegend = 4
        YAxis:
          Label = {$mappFramework/Report/Texts/NumRejects}
          NumberOfGridLines = 9
          ItemMaxValue:
            Value = 1500
        [0]:
          Value:
            ProcessVariable = ::ReportMgr:ReportExample.AdvancedReport.OeeLine[0].NumRejects
          ItemColor = 0000FF
          LegendText = {$mappFramework/Report/Texts/Line1LegendText}
        [1]:
          Value:
            ProcessVariable = ::ReportMgr:ReportExample.AdvancedReport.OeeLine[1].NumRejects
          ItemColor = 008080
          LegendText = {$mappFramework/Report/Texts/Line2LegendText}
        [2]:
          Value:
            ProcessVariable = ::ReportMgr:ReportExample.AdvancedReport.OeeLine[2].NumRejects
          ItemColor = 33CC00
          LegendText = {$mappFramework/Report/Texts/Line3LegendText}
      [3]:
        Name = LineOnePie
        ChartStyle = Default
        TextStyle = ChartText
        ShowLegend = 4
        [0]:
          Value:
            ProcessVariable = ::ReportMgr:ReportExample.AdvancedReport.OeeLine[0].PartsMade
          ItemBackColor = FF9900
          LegendText = {$mappFramework/Report/Texts/PartsMade}
        [1]:
          Value:
            ProcessVariable = ::ReportMgr:ReportExample.AdvancedReport.OeeLine[0].NumRejects
          ItemBackColor = 7F7F7F
          LegendText = {$mappFramework/Report/Texts/NumRejects}
      [4]:
        Name = LineTwoPie
        ChartStyle = Default
        TextStyle = ChartText
        ShowLegend = 4
        [0]:
          Value:
            ProcessVariable = ::ReportMgr:ReportExample.AdvancedReport.OeeLine[1].PartsMade
          ItemBackColor = FF9900
          LegendText = {$mappFramework/Report/Texts/PartsMade}
        [1]:
          Value:
            ProcessVariable = ::ReportMgr:ReportExample.AdvancedReport.OeeLine[1].NumRejects
          ItemBackColor = 7F7F7F
          LegendText = {$mappFramework/Report/Texts/NumRejects}
      [5]:
        Name = LineThreePie
        ChartStyle = Default
        TextStyle = ChartText
        ShowLegend = 4
        [0]:
          Value:
            ProcessVariable = ::ReportMgr:ReportExample.AdvancedReport.OeeLine[2].PartsMade
          ItemBackColor = FF9900
          LegendText = {$mappFramework/Report/Texts/PartsMade}
        [1]:
          Value:
            ProcessVariable = ::ReportMgr:ReportExample.AdvancedReport.OeeLine[2].NumRejects
          ItemBackColor = 7F7F7F
          LegendText = {$mappFramework/Report/Texts/NumRejects}
    Components:
      [0]:
        AlarmHistoryLink = gMpLinkAlarmXHistory
        EmptyListText = {$mappFramework/Report/Texts/EmptyAlarmListText}
        TableStyle = Default
        TextStyle = TableText
        SELECT:
          [0]:
            Column = TimeStamp
            Width = 20
            Heading = SingleText
              Text = {$mappFramework/Report/Texts/TimeStamp}
          [1]:
            Column = Code
            Width = 5
            Heading = SingleText
              Text = {$mappFramework/Report/Texts/Code}
          [2]:
            Width = 15
            Heading = SingleText
              Text = {$mappFramework/Report/Texts/Name}
          [3]:
            Column = Message
            Width = 40
            Heading = SingleText
              Text = {$mappFramework/Report/Texts/Message}
          [4]:
            Column = StateChange
              DisplayAs:
                ActiveText = {$mappFramework/Report/Texts/Activated}
                InactiveText = {$mappFramework/Report/Texts/Deactivated}
                AcknowledgeText = {$mappFramework/Report/Texts/Acknowledged}
                UnacknowledgeText = {$mappFramework/Report/Texts/Unacknowledged}
                UpdateText = {$mappFramework/Report/Texts/Updated}
            Width = 20
            Heading = SingleText
              Text = {$mappFramework/Report/Texts/StateChange}
      [1] = AuditTrail
        AuditTrailLink = gMpLinkAuditTrail
        EmptyListText = {$mappFramework/Report/Texts/EmptyAuditListText}
        TableStyle = Default
        TextStyle = TableText
        SELECT:
          [0]:
            Column = evtime
            Width = 20
            Heading = SingleText
              Text = {$mappFramework/Report/Texts/TimeStamp}
          [1]:
            Column = dtext
            Width = 60
            Heading = SingleText
              Text = {$mappFramework/Report/Texts/Text}
          [2]:
            Column = old
            Width = 10
            Heading = SingleText
              Text = {$mappFramework/Report/Texts/OldValue}
          [3]:
            Column = new
            Width = 10
            Heading = SingleText
              Text = {$mappFramework/Report/Texts/NewValue}
    Contents:
      [0]:
        Name = Header
        [0] = Image
          Image = Images\LogoWithTag.jpg
          HorizontalAlign = 2
        [1]:
          Text = {$mappFramework/Report/Texts/AdvancedHeaderText}
          HorizontalAlign = 1
          NewLine = FALSE
          TextStyle = Title
        [2]:
          Text = {$mappFramework/Report/Texts/BatchHeaderText}
          TextStyle = Default
        [3] = EmptyLine
          Size = 20
      [1]:
        Name = Footer
        [0] = PageNumber
          PageNumSnippet = {$mappFramework/Report/Texts/FooterText}
          HorizontalAlign = 2
          NewLine = FALSE
          TextStyle = Description
      [2]:
        Name = Intro
        [0]:
          Text = {$mappFramework/Report/Texts/IntroText}
          TextStyle = Default
        [1] = EmptyLine
          Size = 20
      [3]:
        Name = DailySummary
        [0] = Line
          LineStyle = Default
        [1] = EmptyLine
          Size = 20
        [2]:
          Text = {$mappFramework/Report/Texts/DailySummaryText}
          HorizontalAlign = 1
          TextStyle = Description
        [3] = EmptyLine
          Size = 20
        [4] = Table
          Table = DailySummary
          HorizontalAlign = 1
        [5] = EmptyLine
          Size = 20
      [4]:
        Name = ProductsChart
        [0] = Line
          LineStyle = Default
        [1] = EmptyLine
          Size = 20
        [2]:
          Text = {$mappFramework/Report/Texts/ProductsChartText}
          HorizontalAlign = 1
          TextStyle = Description
        [3] = EmptyLine
          Size = 20
        [4] = Chart
          Chart = PartsBarChart
          Width = 60
          Height = UserDefined
            Scaling = 35
          HorizontalAlign = 1
        [5] = EmptyLine
          Size = 20
      [5]:
        Name = RejectsChart
        [0]:
          Text = {$mappFramework/Report/Texts/RejectsChartText}
          HorizontalAlign = 1
          TextStyle = Description
        [1] = EmptyLine
          Size = 20
        [2] = Chart
          Chart = RejectsBarChart
          Width = 60
          Height = UserDefined
            Scaling = 35
          HorizontalAlign = 1
        [3] = EmptyLine
          Size = 20
      [6]:
        Name = LineOnePie
        [0]:
          Text = {$mappFramework/Report/Texts/Line1PieText}
          HorizontalAlign = 1
          TextStyle = Description
        [1] = Chart
          Chart = LineOnePie
          Width = 60
          Height = UserDefined
            Scaling = 28
          HorizontalAlign = 1
        [2] = EmptyLine
          Size = 20
      [7]:
        Name = LineTwoPie
        [0]:
          Text = {$mappFramework/Report/Texts/Line2PieText}
          HorizontalAlign = 1
          TextStyle = Description
        [1] = Chart
          Chart = LineTwoPie
          Width = 60
          Height = UserDefined
            Scaling = 28
          HorizontalAlign = 1
        [2] = EmptyLine
          Size = 20
      [8]:
        Name = LineThreePie
        [0]:
          Text = {$mappFramework/Report/Texts/Line3PieText}
          HorizontalAlign = 1
          TextStyle = Description
        [1] = Chart
          Chart = LineThreePie
          Width = 60
          Height = UserDefined
            Scaling = 28
          HorizontalAlign = 1
      [9]:
        Name = TemperatureChart
        [0] = Line
          LineStyle = Default
        [1] = EmptyLine
          Size = 20
        [2]:
          Text = {$mappFramework/Report/Texts/TempChartText}
          HorizontalAlign = 1
          TextStyle = Description
        [3] = EmptyLine
          Size = 20
        [4] = Chart
          Chart = TempLineChart
          Height = UserDefined
            Scaling = 80
          HorizontalAlign = 1
        [5] = EmptyLine
          Size = 20
      [10]:
        Name = Alarms
        [0] = Line
          LineStyle = Default
        [1] = Component
          Component = AlarmHistory
        [2] = EmptyLine
          Size = 20
      [11]:
        Name = Audits
        [0] = Line
          LineStyle = Default
        [1] = Component
          Component = AuditTrail
        [2] = EmptyLine
          Size = 20
      [12]:
        Name = OperatorSignature
        [0] = EmptyLine
          Size = 20
        [1] = EmptyLine
          Size = 20
        [2]:
          Text = {$mappFramework/Report/Texts/OperatorSignature}
          TextStyle = Default
    Reports:
      [0]:
        Name = AdvancedReport
        PageLayout = Default
        Header = Header
        Footer = Footer
        [0]:
          Heading:
            Text = 
            HorizontalAlign = 1
            TextStyle = Default
          [0]:
            Content = Intro
        [1]:
          Heading:
            Text = {$mappFramework/Report/Texts/DailySummaryHeading}
            TextStyle = Default
          [0]:
            Content = DailySummary
        [2]:
          StartOnNewPage = TRUE
          Heading:
            Text = {$mappFramework/Report/Texts/PartsAndRejectsHeading}
            TextStyle = Default
          [0]:
            Content = ProductsChart
        [3]:
          [0]:
            Content = RejectsChart
        [4]:
          StartOnNewPage = TRUE
          Heading:
            Text = {$mappFramework/Report/Texts/PartsAndRejectsHeading}
            TextStyle = Default
          [0]:
            Content = LineOnePie
        [5]:
          Heading:
            Text = 
            TextStyle = Default
          [0]:
            Content = LineTwoPie
        [6]:
          Heading:
            Text = 
            TextStyle = Default
          [0]:
            Content = LineThreePie
        [7]:
          StartOnNewPage = TRUE
          Heading:
            Text = {$mappFramework/Report/Texts/TempSamplesHeading}
            TextStyle = Default
          [0]:
            Content = TemperatureChart
        [8]:
          StartOnNewPage = TRUE
          Heading:
            Text = {$mappFramework/Report/Texts/AlarmHeading}
            TextStyle = Default
          [0]:
            Content = Alarms
        [9]:
          StartOnNewPage = TRUE
          Heading:
            Text = {$mappFramework/Report/Texts/AuditHeading}
            TextStyle = Default
          [0]:
            Content = Audits
        [10]:
          StartOnNewPage = TRUE
          [0]:
            Content = OperatorSignature
  Alarms = MpAlarmX
    mapp.AlarmX.Core.Configuration:
      [0]:
        Message = {$mappFramework/Report/Alarms/GenerateFailed}
```

### Cfg_21CFR1.mpreportcore - PC/mappServices/Report/Cfg_21CFR1.mpreportcore
```
Element gMpLinkReport_21CFR1 (Type=mpreportcore)
  MpReport:
    Settings:
      ResourceDeviceName = mappReportFiles
      LanguageDependent:
        [0]:
          Language = en
        [1]:
          Language = de
    PageLayouts:
      [0]:
        Name = Default
        Orientation = 2
        Margins = 2
    Styles:
      Text:
        [0]:
          Name = Default
        [1]:
          Name = Title
          Size = 20
        [2]:
          Name = Description
          Color = FF9900
        [3]:
          Name = TableText
          NumberOfDecimalPlaces = 2
        [4]:
          Name = ChartText
          NumberOfDecimalPlaces = 2
      Table:
        [0]:
          Name = Default
        [1]:
          Name = ThickBorder_Blue_HighPadding
          BorderWidth = 3
          Color = 0000FF
          Padding = 3
      Line:
        [0]:
          Name = Default
        [1]:
          Name = ThickOrangeLine
          Width = 5
          Color = FF9900
      Chart:
        PieChart:
          [0]:
            Name = Default
          [1]:
            Name = ColorPieChart
            BackColor = 008080
            BorderWidth = 3
            BorderColor = 33CC00
            Padding = 3
        LineChart:
          [0]:
            Name = Default
          [1]:
            Name = ColorLineChart
            BackColor = 008080
            BorderWidth = 3
            BorderColor = 33CC00
            Padding = 3
            GraphBackColor = C0C0C0
            GraphBorderWidth = 3
            GraphBorderColor = 808000
            GridLineWidth = 3
            GridLineColor = 7F7F7F
        BarChart:
          [0]:
            Name = Default
          [1]:
            Name = ColorBarChart
            BackColor = 008080
            BorderWidth = 3
            BorderColor = 33CC00
            Padding = 3
            ItemGapWidth = 3
            GraphBackColor = C0C0C0
            GraphBorderWidth = 3
            GraphBorderColor = 808000
            GridLineWidth = 3
            GridLineColor = 7F7F7F
    Tables:
      [0]:
        Name = DailySummary
        TableStyle = Default
        TextStyle = TableText
        [0]:
          [0] = TextId
            Source = {$MpReport/Ex/RunTime}
            Width = 20
            HorizontalAlign = 1
          [1] = TextId
            Source = {$MpReport/Ex/UpTime}
            Width = 20
            HorizontalAlign = 1
          [2] = TextId
            Source = {$MpReport/Ex/DownTime}
            Width = 20
            HorizontalAlign = 1
          [3] = TextId
            Source = {$MpReport/Ex/PartsMade}
            Width = 20
            HorizontalAlign = 1
          [4] = TextId
            Source = {$MpReport/Ex/PPM}
            Width = 10
            HorizontalAlign = 1
          [5] = TextId
            Source = {$MpReport/Ex/NumRejects}
            Width = 10
            HorizontalAlign = 1
        [1]:
          [0] = ValueId
            Value:
              ProcessVariable = ::ReportMgr:ReportExample.SimpleReport.Line_OEE[0].RunTime
            Width = 20
          [1] = ValueId
            Value:
              ProcessVariable = ::ReportMgr:ReportExample.SimpleReport.Line_OEE[0].UpTime
            Width = 20
          [2] = ValueId
            Value:
              ProcessVariable = ::ReportMgr:ReportExample.SimpleReport.Line_OEE[0].DownTime
            Width = 20
          [3] = ValueId
            Value:
              ProcessVariable = ::ReportMgr:ReportExample.SimpleReport.Line_OEE[0].PartsMade
            Width = 20
            HorizontalAlign = 2
          [4] = ValueId
            Value:
              ProcessVariable = ::ReportMgr:ReportExample.SimpleReport.Line_OEE[0].PPM
            Width = 10
            HorizontalAlign = 2
          [5] = ValueId
            Value:
              ProcessVariable = ::ReportMgr:ReportExample.SimpleReport.Line_OEE[0].NumRejects
            Width = 10
            HorizontalAlign = 2
        [2]:
          [0] = ValueId
            Value:
              ProcessVariable = ::ReportMgr:ReportExample.SimpleReport.Line_OEE[1].RunTime
            Width = 20
          [1] = ValueId
            Value:
              ProcessVariable = ::ReportMgr:ReportExample.SimpleReport.Line_OEE[1].UpTime
            Width = 20
          [2] = ValueId
            Value:
              ProcessVariable = ::ReportMgr:ReportExample.SimpleReport.Line_OEE[1].DownTime
            Width = 20
          [3] = ValueId
            Value:
              ProcessVariable = ::ReportMgr:ReportExample.SimpleReport.Line_OEE[1].PartsMade
            Width = 20
            HorizontalAlign = 2
          [4] = ValueId
            Value:
              ProcessVariable = ::ReportMgr:ReportExample.SimpleReport.Line_OEE[1].PPM
            Width = 10
            HorizontalAlign = 2
          [5] = ValueId
            Value:
              ProcessVariable = ::ReportMgr:ReportExample.SimpleReport.Line_OEE[1].NumRejects
            Width = 10
            HorizontalAlign = 2
        [3]:
          [0] = ValueId
            Value:
              ProcessVariable = ::ReportMgr:ReportExample.SimpleReport.Line_OEE[2].RunTime
            Width = 20
          [1] = ValueId
            Value:
              ProcessVariable = ::ReportMgr:ReportExample.SimpleReport.Line_OEE[2].UpTime
            Width = 20
          [2] = ValueId
            Value:
              ProcessVariable = ::ReportMgr:ReportExample.SimpleReport.Line_OEE[2].DownTime
            Width = 20
          [3] = ValueId
            Value:
              ProcessVariable = ::ReportMgr:ReportExample.SimpleReport.Line_OEE[2].PartsMade
            Width = 20
            HorizontalAlign = 2
          [4] = ValueId
            Value:
              ProcessVariable = ::ReportMgr:ReportExample.SimpleReport.Line_OEE[2].PPM
            Width = 10
            HorizontalAlign = 2
          [5] = ValueId
            Value:
              ProcessVariable = ::ReportMgr:ReportExample.SimpleReport.Line_OEE[2].NumRejects
            Width = 10
            HorizontalAlign = 2
    Charts:
      [0] = LineChart
        Name = TempLineChart
        Heading = SingleText
          Text = {$MpReport/Ex/TempLineChartHeading}
          HorizontalAlign = 1
          TextStyle = Default
        ChartStyle = Default
        TextStyle = ChartText
        ShowLegend = 4
        Y[0]:
          Name = Temperature
          Label = {$MpReport/Ex/TempChartYAxisLabel}
          NumberOfGridLines = 9
          GraphMinValue:
            Value = 10
          GraphMaxValue:
            Value = 110
        XAxis:
          ProcessVariable = ::ReportMgr:ReportExample.SimpleReport.Line_OEE[0].TempSamples.TimeStamp
        [0]:
          YAxis = Temperature
          Value:
            ProcessVariable = ::ReportMgr:ReportExample.SimpleReport.Line_OEE[0].TempSamples.Temp
          LegendText = {$MpReport/Ex/Line1LegendText}
        [1]:
          YAxis = Temperature
          Value:
            ProcessVariable = ::ReportMgr:ReportExample.SimpleReport.Line_OEE[1].TempSamples.Temp
          LineColor = 33CC00
          LegendText = {$MpReport/Ex/Line2LegendText}
        [2]:
          YAxis = Temperature
          Value:
            ProcessVariable = ::ReportMgr:ReportExample.SimpleReport.Line_OEE[2].TempSamples.Temp
          LineColor = 0000FF
          LegendText = {$MpReport/Ex/Line3LegendText}
      [1] = BarChart
        Name = PartsBarChart
        ChartStyle = Default
        TextStyle = ChartText
        ShowLegend = 4
        YAxis:
          Label = {$MpReport/Ex/PartsMade}
          NumberOfGridLines = 9
          ItemMaxValue:
            Value = 100000
        [0]:
          Value:
            ProcessVariable = ::ReportMgr:ReportExample.SimpleReport.Line_OEE[0].PartsMade
          ItemColor = 0000FF
          LegendText = {$MpReport/Ex/Line1LegendText}
        [1]:
          Value:
            ProcessVariable = ::ReportMgr:ReportExample.SimpleReport.Line_OEE[1].PartsMade
          ItemColor = 008080
          LegendText = {$MpReport/Ex/Line2LegendText}
        [2]:
          Value:
            ProcessVariable = ::ReportMgr:ReportExample.SimpleReport.Line_OEE[2].PartsMade
          ItemColor = 33CC00
          LegendText = {$MpReport/Ex/Line3LegendText}
      [2] = BarChart
        Name = RejectsBarChart
        ChartStyle = Default
        TextStyle = ChartText
        ShowLegend = 4
        YAxis:
          Label = {$MpReport/Ex/NumRejects}
          NumberOfGridLines = 9
          ItemMaxValue:
            Value = 1500
        [0]:
          Value:
            ProcessVariable = ::ReportMgr:ReportExample.SimpleReport.Line_OEE[0].NumRejects
          ItemColor = 0000FF
          LegendText = {$MpReport/Ex/Line1LegendText}
        [1]:
          Value:
            ProcessVariable = ::ReportMgr:ReportExample.SimpleReport.Line_OEE[1].NumRejects
          ItemColor = 008080
          LegendText = {$MpReport/Ex/Line2LegendText}
        [2]:
          Value:
            ProcessVariable = ::ReportMgr:ReportExample.SimpleReport.Line_OEE[2].NumRejects
          ItemColor = 33CC00
          LegendText = {$MpReport/Ex/Line3LegendText}
      [3]:
        Name = LineOnePie
        ChartStyle = Default
        TextStyle = ChartText
        ShowLegend = 4
        [0]:
          Value:
            ProcessVariable = ::ReportMgr:ReportExample.SimpleReport.Line_OEE[0].PartsMade
          ItemBackColor = FF9900
          LegendText = {$MpReport/Ex/PartsMade}
        [1]:
          Value:
            ProcessVariable = ::ReportMgr:ReportExample.SimpleReport.Line_OEE[0].NumRejects
          ItemBackColor = 7F7F7F
          LegendText = {$MpReport/Ex/NumRejects}
      [4]:
        Name = LineTwoPie
        ChartStyle = Default
        TextStyle = ChartText
        ShowLegend = 4
        [0]:
          Value:
            ProcessVariable = ::ReportMgr:ReportExample.SimpleReport.Line_OEE[1].PartsMade
          ItemBackColor = FF9900
          LegendText = {$MpReport/Ex/PartsMade}
        [1]:
          Value:
            ProcessVariable = ::ReportMgr:ReportExample.SimpleReport.Line_OEE[1].NumRejects
          ItemBackColor = 7F7F7F
          LegendText = {$MpReport/Ex/NumRejects}
      [5]:
        Name = LineThreePie
        ChartStyle = Default
        TextStyle = ChartText
        ShowLegend = 4
        [0]:
          Value:
            ProcessVariable = ::ReportMgr:ReportExample.SimpleReport.Line_OEE[2].PartsMade
          ItemBackColor = FF9900
          LegendText = {$MpReport/Ex/PartsMade}
        [1]:
          Value:
            ProcessVariable = ::ReportMgr:ReportExample.SimpleReport.Line_OEE[2].NumRejects
          ItemBackColor = 7F7F7F
          LegendText = {$MpReport/Ex/NumRejects}
    Components:
      [0]:
        AlarmHistoryLink = gMpLinkAlarmXHistory
        EmptyListText = {$MpReport/Ex/EmptyAlarmListText}
        TableStyle = Default
        TextStyle = TableText
        SELECT:
          [0]:
            Column = TimeStamp
            Width = 20
            Heading = SingleText
              Text = {$MpReport/Ex/TimeStamp}
          [1]:
            Column = Code
            Width = 10
            Heading = SingleText
              Text = {$MpReport/Ex/Code}
          [2]:
            Width = 20
            Heading = SingleText
              Text = {$MpReport/Ex/Name}
          [3]:
            Column = Message
            Width = 50
            Heading = SingleText
              Text = {$MpReport/Ex/Message}
        WHERE:
          Connect = 
          [0]
          [1]
          [2]
          [3]
      [1] = AuditTrail
        AuditTrailLink = gMpLinkAuditTrail
        EmptyListText = {$MpReport/Ex/EmptyAuditListText}
        TableStyle = Default
        TextStyle = TableText
        SELECT:
          [0]:
            Column = evtime
            Width = 20
            Heading = SingleText
              Text = {$MpReport/Ex/TimeStamp}
          [1]:
            Column = dtext
            Width = 60
            Heading = SingleText
              Text = {$MpReport/Ex/Text}
          [2]:
            Column = old
            Width = 10
            Heading = SingleText
              Text = {$MpReport/Ex/OldValue}
          [3]:
            Column = new
            Width = 10
            Heading = SingleText
              Text = {$MpReport/Ex/NewValue}
        WHERE:
          Connect = 
          [0]
          [1]
          [2]
          [3]
    Contents:
      [0]:
        Name = Header
        [0] = Image
          Image = Images\LogoWithTag.jpg
          HorizontalAlign = 2
        [1]:
          Text = {$MpReport/Ex/HeaderText_21CFR1}
          HorizontalAlign = 1
          NewLine = FALSE
          TextStyle = Title
        [2]:
          Text = {$MpReport/Ex/BatchHeaderText}
          TextStyle = Default
        [3] = EmptyLine
          Size = 20
      [1]:
        Name = Footer
        [0] = PageNumber
          PageNumSnippet = {$MpReport/Ex/FooterText}
          HorizontalAlign = 2
          NewLine = FALSE
          TextStyle = Description
      [2]:
        Name = Intro
        [0]:
          Text = {$MpReport/Ex/IntroText}
          TextStyle = Default
        [1] = EmptyLine
          Size = 20
      [3]:
        Name = DailySummary
        [0] = Line
          LineStyle = Default
        [1] = EmptyLine
          Size = 20
        [2]:
          Text = {$MpReport/Ex/DailySummaryText}
          HorizontalAlign = 1
          TextStyle = Description
        [3] = EmptyLine
          Size = 20
        [4] = Table
          Table = DailySummary
          HorizontalAlign = 1
        [5] = EmptyLine
          Size = 20
      [4]:
        Name = ProductsChart
        [0] = Line
          LineStyle = Default
        [1] = EmptyLine
          Size = 20
        [2]:
          Text = {$MpReport/Ex/ProductsChartText}
          HorizontalAlign = 1
          TextStyle = Description
        [3] = EmptyLine
          Size = 20
        [4] = Chart
          Chart = PartsBarChart
          Width = 60
          Height = UserDefined
            Scaling = 35
          HorizontalAlign = 1
        [5] = EmptyLine
          Size = 20
      [5]:
        Name = RejectsChart
        [0]:
          Text = {$MpReport/Ex/RejectsChartText}
          HorizontalAlign = 1
          TextStyle = Description
        [1] = EmptyLine
          Size = 20
        [2] = Chart
          Chart = RejectsBarChart
          Width = 60
          Height = UserDefined
            Scaling = 35
          HorizontalAlign = 1
        [3] = EmptyLine
          Size = 20
      [6]:
        Name = LineOnePie
        [0]:
          Text = {$MpReport/Ex/Line1PieText}
          HorizontalAlign = 1
          TextStyle = Description
        [1] = Chart
          Chart = LineOnePie
          Width = 60
          Height = UserDefined
            Scaling = 28
          HorizontalAlign = 1
        [2] = EmptyLine
          Size = 20
      [7]:
        Name = LineTwoPie
        [0]:
          Text = {$MpReport/Ex/Line2PieText}
          HorizontalAlign = 1
          TextStyle = Description
        [1] = Chart
          Chart = LineTwoPie
          Width = 60
          Height = UserDefined
            Scaling = 28
          HorizontalAlign = 1
        [2] = EmptyLine
          Size = 20
      [8]:
        Name = LineThreePie
        [0]:
          Text = {$MpReport/Ex/Line3PieText}
          HorizontalAlign = 1
          TextStyle = Description
        [1] = Chart
          Chart = LineThreePie
          Width = 60
          Height = UserDefined
            Scaling = 28
          HorizontalAlign = 1
      [9]:
        Name = TemperatureChart
        [0] = Line
          LineStyle = Default
        [1] = EmptyLine
          Size = 20
        [2]:
          Text = {$MpReport/Ex/TempChartText}
          HorizontalAlign = 1
          TextStyle = Description
        [3] = EmptyLine
          Size = 20
        [4] = Chart
          Chart = TempLineChart
          Height = UserDefined
            Scaling = 80
          HorizontalAlign = 1
        [5] = EmptyLine
          Size = 20
      [10]:
        Name = Alarms
        [0] = Line
          LineStyle = Default
        [1] = Component
          Component = AlarmHistory
        [2] = EmptyLine
          Size = 20
      [11]:
        Name = Audits
        [0] = Line
          LineStyle = Default
        [1] = Component
          Component = AuditTrail
        [2] = EmptyLine
          Size = 20
      [12]:
        Name = OperatorSignature
        [0] = EmptyLine
          Size = 20
        [1] = EmptyLine
          Size = 20
        [2]:
          Text = {$MpReport/Ex/OperatorSignature}
          TextStyle = Default
    Reports:
      [0]:
        Name = Report_21CFR1
        PageLayout = Default
        Header = Header
        Footer = Footer
        [0]:
          Heading:
            Text = 
            HorizontalAlign = 1
            TextStyle = Default
          [0]:
            Content = Intro
        [1]:
          Heading:
            Text = {$MpReport/Ex/DailySummaryHeading}
            TextStyle = Default
          [0]:
            Content = DailySummary
        [2]:
          StartOnNewPage = TRUE
          Heading:
            Text = {$MpReport/Ex/PartsAndRejectsHeading}
            TextStyle = Default
          [0]:
            Content = ProductsChart
        [3]:
          [0]:
            Content = RejectsChart
        [4]:
          StartOnNewPage = TRUE
          Heading:
            Text = {$MpReport/Ex/PartsAndRejectsHeading}
            TextStyle = Default
          [0]:
            Content = LineOnePie
        [5]:
          Heading:
            Text = 
            TextStyle = Default
          [0]:
            Content = LineTwoPie
        [6]:
          Heading:
            Text = 
            TextStyle = Default
          [0]:
            Content = LineThreePie
        [7]:
          StartOnNewPage = TRUE
          Heading:
            Text = {$MpReport/Ex/TempSamplesHeading}
            TextStyle = Default
          [0]:
            Content = TemperatureChart
        [8]:
          StartOnNewPage = TRUE
          Heading:
            Text = {$MpReport/Ex/AlarmHeading}
            TextStyle = Default
          [0]:
            Content = Alarms
        [9]:
          StartOnNewPage = TRUE
          Heading:
            Text = {$MpReport/Ex/AuditHeading}
            TextStyle = Default
          [0]:
            Content = Audits
        [10]:
          StartOnNewPage = TRUE
          [0]:
            Content = OperatorSignature
  Alarms = MpAlarmX
    mapp.AlarmX.Core.Configuration:
      [0]:
        Message = {$Report/Alarms/GenerateFailed}
```

### ReportCfg.mpreportcore - PC/mappServices/Report/ReportCfg.mpreportcore
```
Element gReport (Type=mpreportcore)
  MpReport:
    PageLayouts:
      [0]:
        Name = Default
    Styles:
      Text:
        [0]:
          Name = Default
      Table:
        [0]:
          Name = Default
      Line:
        [0]:
          Name = Default
      Chart:
        PieChart:
          [0]:
            Name = Default
        LineChart:
          [0]:
            Name = Default
        BarChart:
          [0]:
            Name = Default
    Reports:
      [0]:
        PageLayout = Default
        [0]
```

### ReportFile.mpfilemanagerui - PC/mappServices/Report/ReportFile.mpfilemanagerui
```
Element gMpLinkFileManagerUIReport (Type=mpfilemanagerui)
  FileMan:
    CustomizedFileType:
      [0] = .pdf
  Alarms = MpAlarmX
    mapp.AlarmX.Core.Configuration:
      [0]:
        Message = {$File/Alarms/DeviceNotFound}
      [1]:
        Message = {$File/Alarms/AlreadyExisting}
      [2]:
        Message = {$File/Alarms/FileSystemError}
```
